(* IEC 61131-3 sources: Stat_Resistant_AI_Coding/src/plc/project/Station010/SqC_Wp100_Run, 2 files *)

(* ---- declaration.st ---- *)
FUNCTION_BLOCK SqC_Wp100_Run EXTENDS OpconSfcChain
////<OES_INFO Mode="Merge" Areas="1/1" />
////<OES_CODE MergeId="Declaration">{{{
VAR_INPUT
  rUnit : REFERENCE TO Wp100Unit;
END_VAR
////<END_OES_CODE>}}}

VAR_OUTPUT
  /// Results of the completed left, middle and right atomic measurements
  Result : Wp100RunSequenceResultStruct;
END_VAR

VAR
  /// Handle of the locked product-detection soft error
  _eventIndex          : UDINT;
  /// Bit 0 = _100B701 missing, bit 1 = _100B702 missing
  _partSensorFaultMask : BYTE;
END_VAR

(* ---- OnChainFinish.st ---- *)
/// Method is called for only one cycle if chain stops working by any given reason
METHOD PROTECTED OnChainFinish
VAR_INPUT
  Reason: OpconChainFinishReason;
END_VAR

// Call base method first, then reset every child execution owned by this chain.
// AI_HMI_FORCE_TRACE_BEGIN
CASE Reason OF
  OpconChainFinishReason.ERROR:
    Station.ForceTraceAddon.Recorder.Finish(Reason := 4,
      LastForceN := Wp100A104Kistler.Unit.OutImm.ForceAct);
  OpconChainFinishReason.CANCEL:
    Station.ForceTraceAddon.Recorder.Finish(Reason := 3,
      LastForceN := Wp100A104Kistler.Unit.OutImm.ForceAct);
END_CASE
// AI_HMI_FORCE_TRACE_END
SUPER^.OnChainFinish(Reason);

CASE Reason OF
  OpconChainFinishReason.ERROR,
  OpconChainFinishReason.CANCEL,
  OpconChainFinishReason.DONE:
    Wp100.SqS_Run.Execute := FALSE;

    IF ( _eventIndex <> 0 )
    THEN
      IF ( UnlockEvent(
           Class := OpconEventClass.SOFTERROR,
           Index := _eventIndex
         ) )
      THEN
        IF ( ClearEvent(
             Class := OpconEventClass.SOFTERROR,
             Index := _eventIndex
           ) )
        THEN
          _eventIndex := 0;
        END_IF
      END_IF
    END_IF

    _partSensorFaultMask := 0;

    IF ( Reason <> OpconChainFinishReason.DONE )
    THEN
      Station._AutoInfoline := AutoInfoLineEnum.USER_INFO_TEXT_CLEAR;
    END_IF

  ELSE
    ; // do nothing
END_CASE
